PROGRAM P01_AnalogScaling
VAR
END_VAR

// NETWORK 1

END_PROGRAM

(* stored: Version 1.1.0.1
   POU P01_AnalogScaling: Id {a513cc6b-23dc-4082-bd01-a08684514783}, SpecialFunc None *)
